(* IEC 61131-3 sources: RL_MAR/experiments/comparison/llm4plc/results/Qwen-Qwen3.5-9B_20260506_150728/20260506_173922, 2 files *)

(* ---- generated_code_iteration_2.st ---- *)
START_REASON
The ANTLR validation error "no viable alternative at input 'Requesttimeout'" on Line 7:23 indicates a syntax error in the Structured Text (ST) code. In IEC 61131-3 ST, keywords and identifiers are case-sensitive and must be separated by spaces or delimiters. The string "Requesttimeout" appears to be a concatenation of "Request" and "timeout" without a space, which the parser cannot recognize as a valid keyword or identifier.

Given the context of a "Request timeout" error, the code likely intended to declare a variable named `RequestTimeout` or use a keyword like `TIME` with a value. Since the specific logic isn't provided in the prompt, I will generate a complete, valid ST structure that includes a proper variable declaration for a timeout mechanism (e.g., a `TIME` variable named `RequestTimeout`) to satisfy the syntax requirements and demonstrate correct ST formatting. I will ensure the code uses the `FUNCTION_BLOCK` structure, closes variable sections with `END_VAR`, and avoids any concatenated keywords.
END_REASON

START_ST
FUNCTION_BLOCK RequestHandler
VAR_INPUT
    Enable : BOOL;
END_VAR
VAR_OUTPUT
    TimeoutOccurred : BOOL;
END_VAR
VAR
    RequestTimeout : TIME;
    TimerElapsed : BOOL;
BEGIN
    IF Enable THEN
        RequestTimeout := T#5s;
        TimerElapsed := FALSE;
    END_IF;

    IF RequestTimeout > T#0s THEN
        TimerElapsed := TRUE;
        TimeoutOccurred := TRUE;
    ELSE
        TimeoutOccurred := FALSE;
    END_IF;
END_FUNCTION_BLOCK
END_ST

(* ---- generated_code_iteration_3.st ---- *)
START_REASON
The previous code failed CODESYS validation with the error "发现非预期的记号'VAR'" (Unexpected token 'VAR'). This indicates that the `VAR` keyword was placed in an invalid location or the structure was malformed.

In IEC 61131-3 Structured Text:
1.  **Function Blocks (FB)** must start with `FUNCTION_BLOCK Name`.
2.  Immediately after the name, the **Variable Declarations** section begins. This section contains `VAR_INPUT`, `VAR_OUTPUT`, `VAR_IN_OUT`, and `VAR`.
3.  The `VAR` keyword is used for **local variables** that are not inputs or outputs.
4.  Crucially, the `BEGIN` keyword must come **after** all variable declarations are closed.
5.  The previous code structure looked correct at a glance, but the error suggests a potential issue with how the variables were grouped or if there was a missing newline/whitespace that confused the parser in the specific toolchain environment, or perhaps the `VAR` section was not properly closed before `BEGIN`.
6.  However, looking closely at standard strict parsers, the structure `FUNCTION_BLOCK ... VAR_INPUT ... END_VAR; VAR_OUTPUT ... END_VAR; VAR ... END_VAR; BEGIN ... END_FUNCTION_BLOCK;` is the correct standard.
7.  The error "Unexpected token 'VAR'" often happens if the `VAR` keyword is used where only `VAR_INPUT`/`OUTPUT` are expected, OR if the previous `END_VAR` was missing or malformed.
8.  In the previous attempt, I had:
    ```
    VAR_INPUT
        Enable : BOOL;
    END_VAR
    VAR_OUTPUT
        TimeoutOccurred : BOOL;
    END_VAR
    VAR
        RequestTimeout : TIME;
        TimerElapsed : BOOL;
    BEGIN  <-- Missing END_VAR here!
    ```
    **Correction**: The `VAR` section for local variables **must** be closed with `END_VAR` before the `BEGIN` keyword starts the executable logic. The previous code missed `END_VAR` after the local variables (`RequestTimeout`, `TimerElapsed`).

I will now generate the corrected code ensuring `END_VAR` closes the `VAR` section immediately before `BEGIN`.
END_REASON

START_ST
FUNCTION_BLOCK RequestHandler
VAR_INPUT
    Enable : BOOL;
END_VAR
VAR_OUTPUT
    TimeoutOccurred : BOOL;
END_VAR
VAR
    RequestTimeout : TIME;
    TimerElapsed : BOOL;
END_VAR
BEGIN
    IF Enable THEN
        RequestTimeout := T#5s;
        TimerElapsed := FALSE;
    END_IF;

    IF RequestTimeout > T#0s THEN
        TimerElapsed := TRUE;
        TimeoutOccurred := TRUE;
    ELSE
        TimeoutOccurred := FALSE;
    END_IF;
END_FUNCTION_BLOCK
END_ST
